(* CoDeSys 2.3.9.42 project: pidd.pro *)
(* Libraries: C:\Users\bnm\Desktop\oscat_basic_333.lib 25.5.18 09:12:18, Util.lib 18.5.10 15:14:28, Standard.lib 4.10.05 11:14:46, IecSfc.lib 13.4.06 15:51:28, SYSLIBCALLBACK.LIB 26.9.08 15:43:52 *)

(* POU PLC_PRG, CFC *)
PROGRAM PLC_PRG
VAR
	PID:CTRL_PID;
	SIG:REAL;
	INPUT:REAL;
	TEMP:REAL;
	TEMPO:REAL;
	KP:REAL;
	TN:REAL;
	TV:REAL;
	SIG_:REAL;
	In_rt2: LIN_TRAFO;
	In_tr1: LIN_TRAFO;
	In_rt3: LIN_TRAFO;
END_VAR
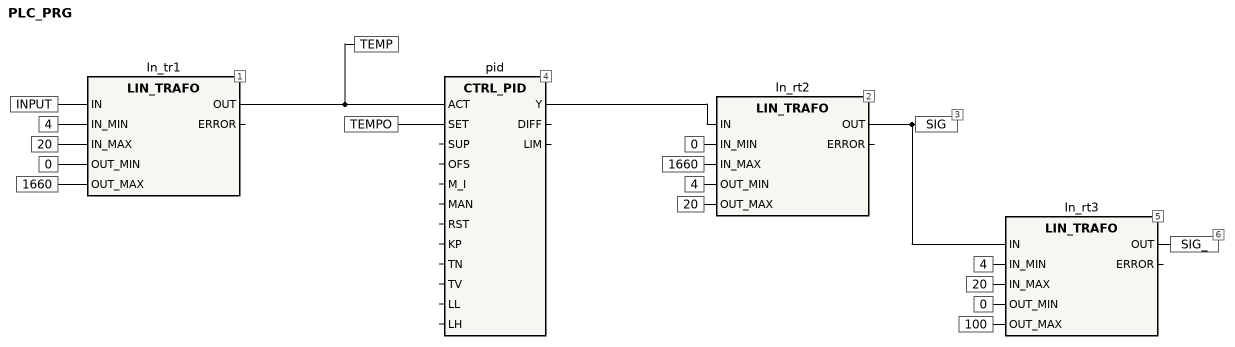
_CFC_ (* Continuous Function Chart, elements in execution order *)
#0 TEMP <= #1.OUT
#1 In_tr1:LIN_TRAFO(IN: INPUT, IN_MIN: 4, IN_MAX: 20, OUT_MIN: 0, OUT_MAX: 1660)
#2 In_rt2:LIN_TRAFO(IN: #4.Y, IN_MIN: 0, IN_MAX: 1660, OUT_MIN: 4, OUT_MAX: 20)
#3 SIG <= #2.OUT
#4 pid:CTRL_PID(ACT: #1.OUT, SET: TEMPO, SUP: -, OFS: -, M_I: -, MAN: -, RST: -, KP: -, TN: -, TV: -, LL: -, LH: -)
#5 In_rt3:LIN_TRAFO(IN: #2.OUT, IN_MIN: 4, IN_MAX: 20, OUT_MIN: 0, OUT_MAX: 100)
#6 SIG_ <= #5.OUT
_END_CFC_
(* the same logic as Structured Text *)
TEMP := In_tr1.OUT;
In_tr1(IN := INPUT, IN_MIN := 4, IN_MAX := 20, OUT_MIN := 0, OUT_MAX := 1660);
In_rt2(IN := pid.Y, IN_MIN := 0, IN_MAX := 1660, OUT_MIN := 4, OUT_MAX := 20);
SIG := In_rt2.OUT;
pid(ACT := In_tr1.OUT, SET := TEMPO);
In_rt3(IN := In_rt2.OUT, IN_MIN := 4, IN_MAX := 20, OUT_MIN := 0, OUT_MAX := 100);
SIG_ := In_rt3.OUT;
END_PROGRAM

(* Visualisation Dima
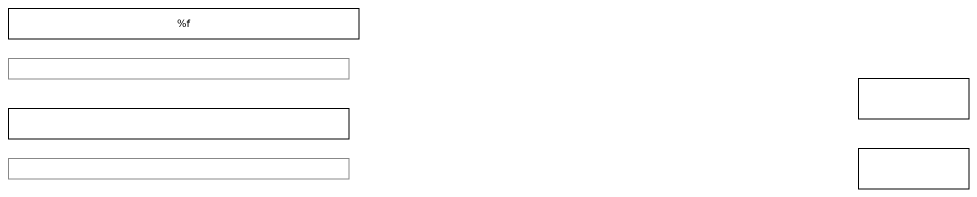
rectangle at (130,30)-(481,61): text "%f"; shows PLC_PRG.TEMP
rectangle at (980,100)-(1091,141): shows PLC_PRG.TV; editable 0..100
rectangle at (980,170)-(1091,211): shows PLC_PRG.TN; editable 0..100
3 more shapes without text or variables
3 elements of other kinds (tables, trends, ...) not read
*)
